TYPE E_StepSubPhase : (
    STEP_SUBPHASE_NONE := 0,
    STEP_SUBPHASE_ENTRY := 10,
    STEP_SUBPHASE_RAMP_PROCESS := 20,
    STEP_SUBPHASE_END_CHECK := 30,
    STEP_SUBPHASE_BRAKE_COMPRESSION := 40,
    STEP_SUBPHASE_VALID_FORCE_HOLD := 50
); END_TYPE

(* stored: Version 1.1.0.1
   DUT E_StepSubPhase: Id {E3000000-0000-4000-8000-000000000009} *)
